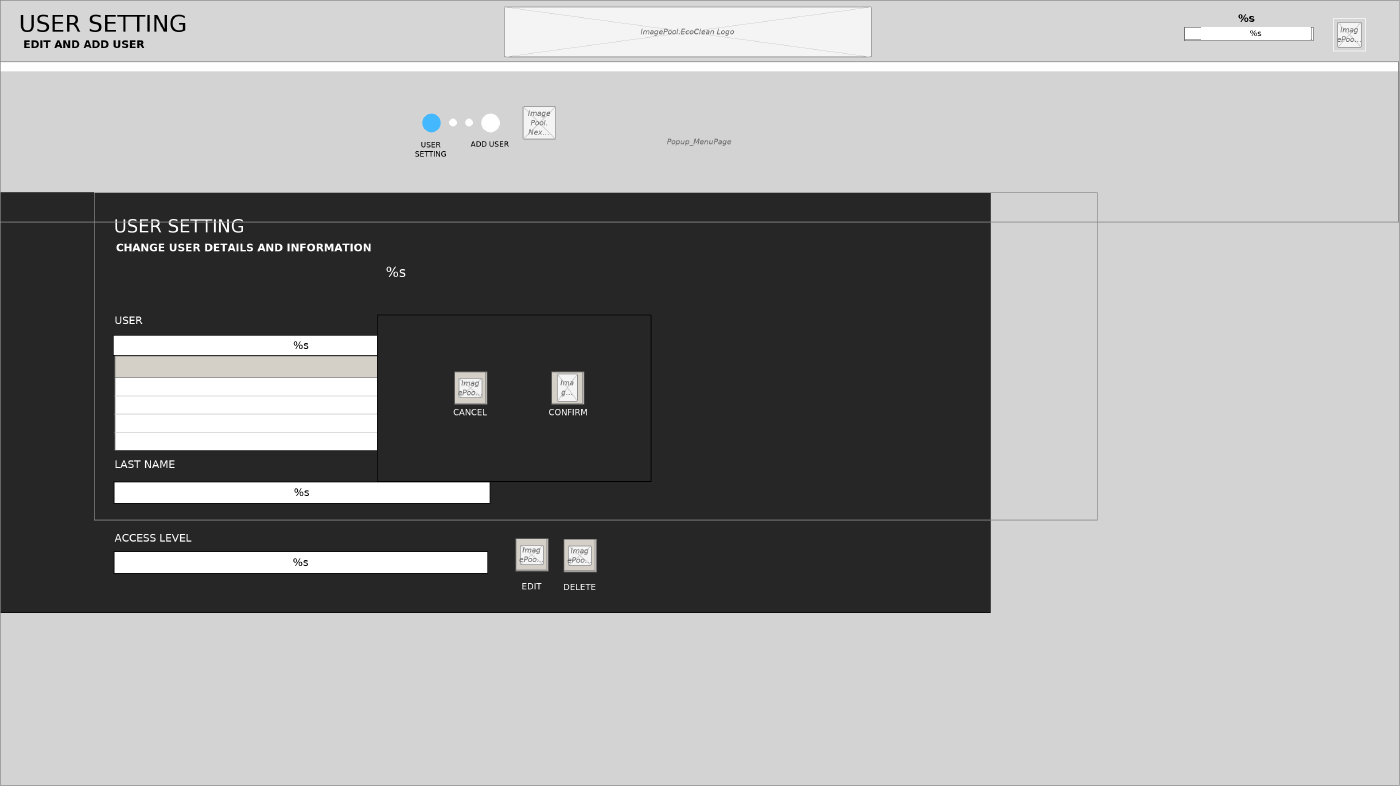
VISUALIZATION UserSetting_Page  // 1920x1079
    Rectangle (0,98 1920x981)
    Rectangle (0,63 1920x26)
        p3528305787: HMI_Ctrl.ANIMATION3
    Rectangle (0,0 1919x85)
    Label (23,6 310x53), "USER SETTING"
    Label (29,49 320x24), "EDIT AND ADD USER"
    Group (1828,25 45x45)
        OnMouseClick: toggle HMI_Ctrl.MenuButton
        RoundedRectangle (0,0 45x45), colour toggle: HMI_Ctrl.MenuButton
        Image (6,5 33x35), image: ImagePool.Menu Button
    Image (691,9 504x69), image: ImagePool.EcoClean Logo
    Group (1621,14 180x42)
        Rectangle (0,0 177x22), "%s", text variable: DSLocalSystemTimeML.sCurrentDT24Hr_General
        Button (3,23 177x19), image: VisuSymbols.Symbols.AddUser
        Rectangle (26,23 150x18), "%s", text variable: fbHmiTF1800_UserlevelManagement.dsHmiUserStatus_Active.sLoginName
    Rectangle (0,264 1358x577)
    Label (153,284 221x53), "USER SETTING"
    Label (156,321 609x38), "CHANGE USER DETAILS AND INFORMATION"
    Label (154,712 216x53), "ACCESS LEVEL"
    Label (154,611 216x53), "LAST NAME"
    Label (154,409 123x62), "USER"
    Label (154,510 216x53), "FIRST NAME"
    RoundedRectangle (550,151 162x35)
    Ellipse (579,156 25x25)
    Ellipse (660,156 25x25)
    Ellipse (616,163 10x10)
    Ellipse (638,163 10x10)
    Label (559,186 64x39), "USER SETTING"
    Label (640,186 64x24), "ADD USER"
    Image (717,146 45x45), image: ImagePool.Next Button
        OnMouseClick: change screen: AddNewUser_Page
    Group (699,739 60x88)
        toggle bUM_EditPB
        OnMouseDown: toggle bUserNameEditPageOn
        OnMouseDown: toggle bUM_EditPB
        Button (8,0 45x45)
        Label (0,44 60x44), "EDIT"
        Image (14,9 32x27), image: ImagePool.Delete User
    Group (155,460 516x28)
        toggle bUserNameLoginPageOn
        Rectangle (0,0 516x28), "%s", text variable: fbHmiTF1800_UserlevelManagement.dsHmiUserReg.ARsLoginName[iUM_SelectedLoginNameId]
        Group (481,0 35x28)
            Rectangle (0,0 40x34)
            Image (4,2 32x32), image: VisuSymbols.Symbols.TriangleDown
    Rectangle (157,557 516x30), "%s", text variable: fbHmiTF1800_UserlevelManagement.dsHmiUserReg.ARsFirstName[iUM_SelectedLoginNameId]
        OnMouseDown: write the text variable via Default
    Rectangle (156,661 516x30), "%s", text variable: fbHmiTF1800_UserlevelManagement.dsHmiUserReg.ARsLastName[iUM_SelectedLoginNameId]
        OnMouseDown: write the text variable via Default
    Textfield (159,359 768x30), "%s", text variable: sMessage
    Table (157,488 512x130), invisible if: NOT bUserNameLoginPageOn, data array: fbHmiTF1800_UserlevelManagement.dsHmiUserReg.ARsLoginName
        p1137915858: iUM_SelectedLoginNameId
        p3854506369: fbHmiTF1800_UserlevelManagement.dsHmiUserReg.ARsLoginName[INDEX]
        p2232123230: Login Name
        Columns.Column.[0].Template: toggle bUserNameLoginPageOn
    Rectangle (156,757 513x30), "%s", text variable: fbHmiTF1800_UserlevelManagement.dsHmiUserReg.ARwsUserGroupName[iUM_SelectedLoginNameId]
    Group (765,740 60x88)
        toggle bUM_DeletePB
        Button (8,0 45x45)
        Label (0,44 60x44), "DELETE"
        Image (14,9 32x27), image: ImagePool.Delete User
    Frame (129,264 1376x450), invisible if: NOT bUserNameEditPageOn
        shows Edit_User()
    Group (517,432 376x229), invisible if: NOT bPageConfirmPageOn
        Rectangle (0,0 376x229)
        Group (230,78 65x68)
            toggle bUM_ConfirmPB
            Button (9,0 45x45)
            Label (0,44 65x24), "CONFIRM"
            Image (17,3 28x38), image: ImagePool.Save Button
        Group (98,78 60x78)
            toggle bUM_ReturnPB
            OnMouseDown: toggle bPageConfirmPageOn
            Button (8,0 45x45)
            Label (0,34 60x44), "CANCEL"
            Image (14,9 32x27), image: ImagePool.Delete User
    Frame (0,84 1918x221), invisible if: HMI_Ctrl.CloseMenuButton
        shows Popup_MenuPage()
END_VISUALIZATION

(* stored: Version 1.1.0.1, ProductVersion 3.1.4024.12
   Visu UserSetting_Page: Id {7f0957c6-e7cb-4824-a9d0-b1ce4daced56} *)
